FUNCTION_BLOCK Mc3MotionHomeTask_SetZeroHere EXTENDS Mc3MotionTask
VAR
	MCSetPosition : Tc3_Mc3Ptp.MC_SetPosition;
END_VAR

{attribute 'monitoring' := 'call'}
PROPERTY Busy : BOOL
GET
Busy := MCSetPosition.Busy;
END_GET
END_PROPERTY

METHOD CyclicLogic
MCSetPosition(Axis := _Axis.Axis);
MCSetPosition.Execute := FALSE;
END_METHOD

{attribute 'monitoring' := 'call'}
PROPERTY Error : BOOL
GET
Error := MCSetPosition.Error;
END_GET
END_PROPERTY

{attribute 'monitoring' := 'call'}
PROPERTY ErrorId : UDINT
GET
ErrorId := MCSetPosition.ErrorID;
END_GET
END_PROPERTY

METHOD Execute : BOOL
IF Axis.Busy OR Axis.Error THEN
	RETURN;
END_IF

MCSetPosition.Execute := TRUE;
Execute				  := TRUE;
END_METHOD

END_FUNCTION_BLOCK

(* stored: Version 1.1.0.1, ProductVersion 3.1.4026.20
   POU Mc3MotionHomeTask_SetZeroHere: Id {725be1b2-6709-422a-931a-48d0125b2bdf}, SpecialFunc None
   Property Busy: Id {98de1fad-0375-4c54-ba65-b5d4d0878a21}
   Get Get: Id {5d64767a-a2d1-4c3b-affa-5af787164406}
   Method CyclicLogic: Id {34dcca4c-9c3b-4a8b-803b-fbf49810501b}
   Property Error: Id {7d4fc4ab-633b-4fe5-8d06-43260ef31148}
   Get Get: Id {a85f9b65-feb0-4ab2-8c7b-47a68056b155}
   Property ErrorId: Id {c48472d5-5f31-416b-a3ed-300f96ce6f3c}
   Get Get: Id {14439ad4-a3bc-4de7-9b16-a78c6f1f34ff}
   Method Execute: Id {bfdc6a1c-d92b-4284-ad51-d564563b4ea9} *)
